// Mitsubishi GX Works2 project: Ehd   PLC: Q02/Q02H

PROGRAM MAIN
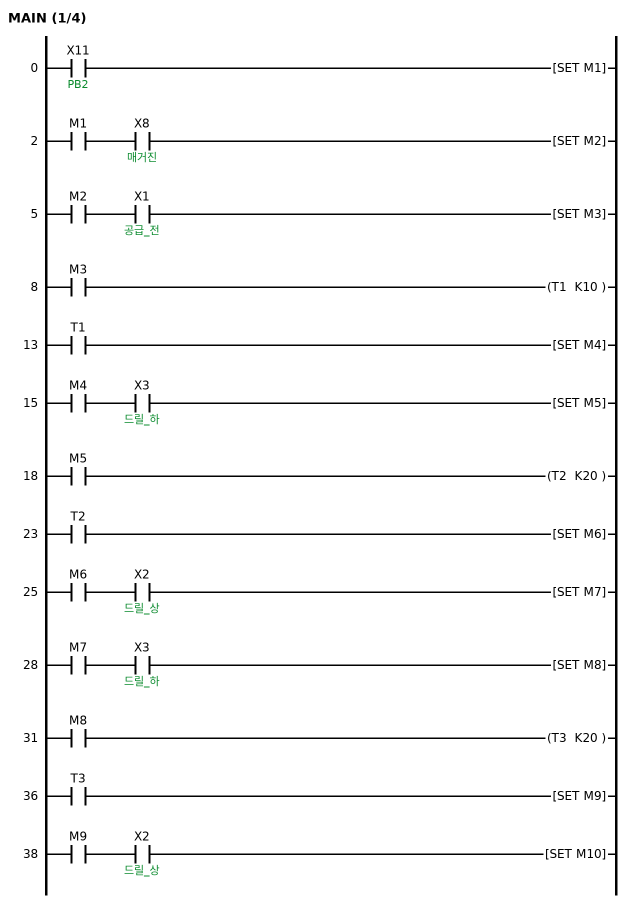
0     LD      X11  ; PB2
      SET     M1
2     LD      M1
      AND     X8  ; 매거진
      SET     M2
5     LD      M2
      AND     X1  ; 공급_전
      SET     M3
8     LD      M3
      OUT     T1 K10
13    LD      T1
      SET     M4
15    LD      M4
      AND     X3  ; 드릴_하
      SET     M5
18    LD      M5
      OUT     T2 K20
23    LD      T2
      SET     M6
25    LD      M6
      AND     X2  ; 드릴_상
      SET     M7
28    LD      M7
      AND     X3  ; 드릴_하
      SET     M8
31    LD      M8
      OUT     T3 K20
36    LD      T3
      SET     M9
38    LD      M9
      AND     X2  ; 드릴_상
      SET     M10
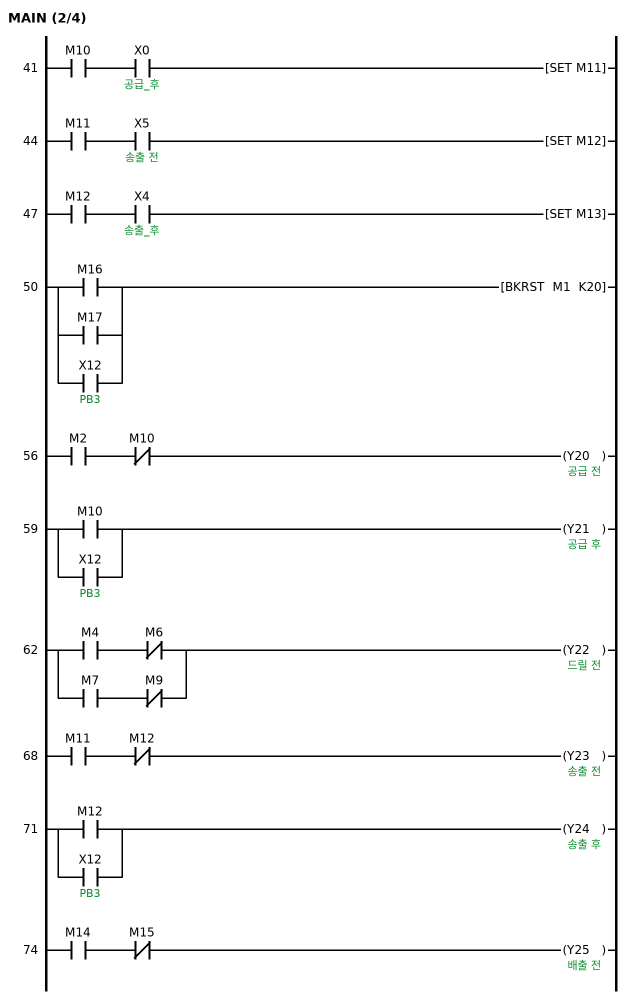
41    LD      M10
      AND     X0  ; 공급_후
      SET     M11
44    LD      M11
      AND     X5  ; 송출 전
      SET     M12
47    LD      M12
      AND     X4  ; 송출_후
      SET     M13
50    LD      M16
      OR      M17
      OR      X12  ; PB3
      BKRST   M1 K20
56    LD      M2
      ANI     M10
      OUT     Y20  ; 공급 전
59    LD      M10
      OR      X12  ; PB3
      OUT     Y21  ; 공급 후
62    LD      M4
      ANI     M6
      LD      M7
      ANI     M9
      ORB
      OUT     Y22  ; 드릴 전
68    LD      M11
      ANI     M12
      OUT     Y23  ; 송출 전
71    LD      M12
      OR      X12  ; PB3
      OUT     Y24  ; 송출 후
74    LD      M14
      ANI     M15
      OUT     Y25  ; 배출 전
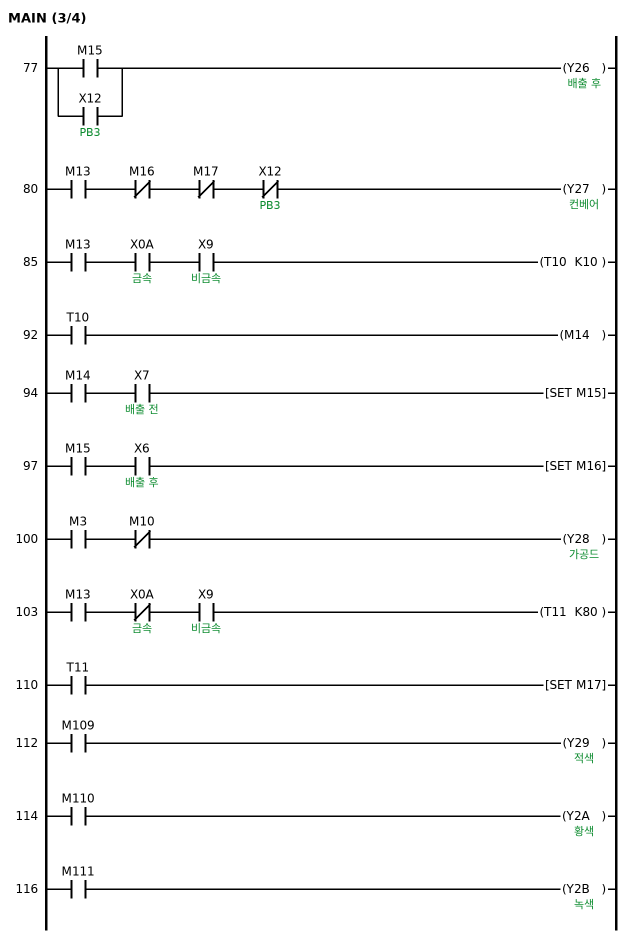
77    LD      M15
      OR      X12  ; PB3
      OUT     Y26  ; 배출 후
80    LD      M13
      ANI     M16
      ANI     M17
      ANI     X12  ; PB3
      OUT     Y27  ; 컨베어
85    LD      M13
      AND     X0A  ; 금속
      AND     X9  ; 비금속
      OUT     T10 K10
92    LD      T10
      OUT     M14
94    LD      M14
      AND     X7  ; 배출 전
      SET     M15
97    LD      M15
      AND     X6  ; 배출 후
      SET     M16
100   LD      M3
      ANI     M10
      OUT     Y28  ; 가공드
103   LD      M13
      ANI     X0A  ; 금속
      AND     X9  ; 비금속
      OUT     T11 K80
110   LD      T11
      SET     M17
112   LD      M109
      OUT     Y29  ; 적색
114   LD      M110
      OUT     Y2A  ; 황색
116   LD      M111
      OUT     Y2B  ; 녹색
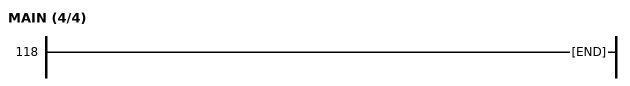
118   END
END_PROGRAM

// device comments not shown above
X10  ; PB1
